{attribute 'call_after_init'}
FUNCTION_BLOCK FB_BPRequestor_Test EXTENDS TcUnit.FB_TestSuite
VAR_INPUT
END_VAR
VAR_OUTPUT
END_VAR
VAR

END_VAR

METHOD PRIVATE BPRequestorSafeGuardFunctionality
VAR_INPUT
END_VAR
VAR
    fbBPR    :    FB_BPRequestor;
END_VAR
TEST('Reset Beam to Safe if Arbiter Faulted');
END_METHOD

END_FUNCTION_BLOCK

(* stored: Version 1.1.0.1, ProductVersion 3.1.4024.0
   POU FB_BPRequestor_Test: Id {c6d3581a-a6af-4d48-bb2e-09f77a3f9bdd}, SpecialFunc None
   Method BPRequestorSafeGuardFunctionality: Id {7127eb59-b63a-41f4-ac69-34ca4a2c3b46} *)
